FUNCTION_BLOCK Reset2
VAR_INPUT
	Execute : BOOL;
END_VAR
VAR_OUTPUT
	Done : BOOL;
END_VAR
VAR
	fbResetAll: FB_ResetAllAxis;
	bResetExecute: BOOL := TRUE;
END_VAR

IF Execute THEN
	Done := FALSE;
	fbResetAll(
		Execute := bResetExecute
	);	
	bResetExecute := TRUE;
	IF fbResetAll.Done THEN
		bResetExecute := FALSE;
		Done := TRUE;
	END_IF
	
ELSE
	Done := FALSE;
	
END_IF

END_FUNCTION_BLOCK

(* stored: Version 1.1.0.1, ProductVersion 3.1.4024.11
   POU Reset2: Id {c18ff4d2-bf50-48ff-89d8-b8e3792d79c2}, SpecialFunc None *)
